TYPE DUT_HIM_DeviceType :
STRUCT
	Ip : STRING(15);
	DeviceType : eDeviceType;
END_STRUCT
END_TYPE

(* stored: Version 1.1.0.1, ProductVersion 3.1.4024.15
   DUT DUT_HIM_DeviceType: Id {be6b483b-3293-4396-9a26-c758a5702c81} *)
